(* IEC 61131-3 sources: VovkPLCRuntime/wasm/node-test/st-tests/st-samples, 20 files *)

(* ---- test_01_variable_declaration.st ---- *)
(* Test 1: Variable Declaration *)
(* Tests basic variable declarations with different IEC 61131-3 types *)

VAR
    counter : INT;
    flag : BOOL;
    temperature : REAL;
END_VAR

(* ---- test_02_var_with_init.st ---- *)
(* Test 2: Variable Declaration with Initialization *)

VAR
    count : INT := 100;
    active : BOOL := TRUE;
    value : REAL := 3.14;
END_VAR

(* ---- test_03_var_at_address.st ---- *)
(* Test 3: Variable Declaration with AT address *)

VAR
    input1 AT %IX0.0 : BOOL;
    output1 AT %QX0.0 : BOOL;
    memory1 AT %MW10 : INT;
END_VAR

(* ---- test_04_all_types.st ---- *)
(* Test 4: All IEC 61131-3 Types *)

VAR
    v_sint : SINT;
    v_int : INT;
    v_dint : DINT;
    v_lint : LINT;
    v_usint : USINT;
    v_uint : UINT;
    v_udint : UDINT;
    v_ulint : ULINT;
    v_byte : BYTE;
    v_word : WORD;
    v_dword : DWORD;
    v_lword : LWORD;
    v_real : REAL;
    v_lreal : LREAL;
END_VAR

(* ---- test_05_assignment.st ---- *)
(* Test 5: Simple Assignment *)

VAR
    a : INT;
    b : INT;
END_VAR

a := 10;
b := a + 5;

(* ---- test_06_arithmetic.st ---- *)
(* Test 6: Arithmetic Operators *)

VAR
    result : INT;
    a : INT := 10;
    b : INT := 3;
END_VAR

result := a + b;
result := a - b;
result := a * b;
result := a / b;
result := a MOD b;

(* ---- test_07_comparison.st ---- *)
(* Test 7: Comparison Operators *)

VAR
    result : BOOL;
    a : INT := 10;
    b : INT := 5;
END_VAR

result := a = b;
result := a <> b;
result := a < b;
result := a > b;
result := a <= b;
result := a >= b;

(* ---- test_08_logical.st ---- *)
(* Test 8: Logical Operators *)

VAR
    result : BOOL;
    a : BOOL := TRUE;
    b : BOOL := FALSE;
END_VAR

result := a AND b;
result := a OR b;
result := a XOR b;
result := NOT a;

(* ---- test_09_bitwise_shift.st ---- *)
(* Test 9: Bitwise Shift Operators *)

VAR
    result : DWORD;
    value : DWORD := 16;
END_VAR

result := value SHL 2;
result := value SHR 1;

(* ---- test_10_if_then.st ---- *)
(* Test 10: Simple IF-THEN-END_IF *)

VAR
    flag : BOOL;
    result : INT;
END_VAR

IF flag THEN
    result := 1;
END_IF;

(* ---- test_11_if_else.st ---- *)
(* Test 11: IF-THEN-ELSE-END_IF *)

VAR
    flag : BOOL;
    result : INT;
END_VAR

IF flag THEN
    result := 1;
ELSE
    result := 0;
END_IF;

(* ---- test_12_if_elsif.st ---- *)
(* Test 12: IF-ELSIF-ELSE-END_IF *)

VAR
    value : INT;
    result : INT;
END_VAR

IF value = 1 THEN
    result := 10;
ELSIF value = 2 THEN
    result := 20;
ELSIF value = 3 THEN
    result := 30;
ELSE
    result := 0;
END_IF;

(* ---- test_13_for_loop.st ---- *)
(* Test 13: Simple FOR Loop *)

VAR
    i : INT;
    sum : INT := 0;
END_VAR

FOR i := 1 TO 10 DO
    sum := sum + i;
END_FOR;

(* ---- test_14_for_loop_by.st ---- *)
(* Test 14: FOR Loop with BY Step *)

VAR
    i : INT;
    count : INT := 0;
END_VAR

FOR i := 0 TO 100 BY 10 DO
    count := count + 1;
END_FOR;

(* ---- test_15_while_loop.st ---- *)
(* Test 15: WHILE Loop *)

VAR
    count : INT := 0;
END_VAR

WHILE count < 10 DO
    count := count + 1;
END_WHILE;

(* ---- test_16_repeat_until.st ---- *)
(* Test 16: REPEAT-UNTIL Loop *)

VAR
    count : INT := 0;
END_VAR

REPEAT
    count := count + 1;
UNTIL count >= 10
END_REPEAT;

(* ---- test_17_exit_break.st ---- *)
(* Test 17: EXIT Statement *)

VAR
    i : INT;
END_VAR

FOR i := 1 TO 100 DO
    IF i = 50 THEN
        EXIT;
    END_IF;
END_FOR;

(* ---- test_18_return.st ---- *)
(* Test 18: RETURN Statement *)

VAR
    flag : BOOL;
END_VAR

IF flag THEN
    RETURN;
END_IF;

(* ---- test_19_case_insensitive.st ---- *)
(* Test 19: Case-Insensitive Keywords *)

var
    Counter : int;
end_var

if Counter = 0 then
    Counter := 1;
end_if;

(* ---- test_20_complex_expression.st ---- *)
(* Test 20: Complex Nested Expression *)

VAR
    result : REAL;
    a : REAL := 1.0;
    b : REAL := 2.0;
    c : REAL := 3.0;
END_VAR

result := (a + b) * (c - a) / (b + c);
